# EPICS alarm handler configuration: alh_files/mgnt_ltu.alhConfig
GROUP NULL MGNT:LTU1:1
   $COMMAND edm -x -eolc -noedit mgnt_ltu1_main.edl

$ALIAS LTU1
$GUIDANCE
ltu Magnet
   Group Name: MGNT:LTU1:1
   Summary PV:  MGNT:LTU1:1:STATSUMY
$END

   INCLUDE MGNT:LTU1:1 ./mgnt_ltu_bend.alhConfig
   INCLUDE MGNT:LTU1:1 ./mgnt_ltu_kick.alhConfig
   INCLUDE MGNT:LTU1:1 ./mgnt_ltu_lgps.alhConfig
   INCLUDE MGNT:LTU1:1 ./mgnt_ltu_quad.alhConfig
   INCLUDE MGNT:LTU1:1 ./mgnt_ltu_xcor.alhConfig
   INCLUDE MGNT:LTU1:1 ./mgnt_ltu_ycor.alhConfig
